// TwinCAT 3 PLC project GetConnectionInfo
// ProgramVersion: 3.1.0.5
// libraries:
//   Tc2_FTP,newest,Beckhoff Automation GmbH
//   Tc2_Standard,newest,Beckhoff Automation GmbH
//   Tc2_System,newest,Beckhoff Automation GmbH
//   Tc3_Module,newest,Beckhoff Automation GmbH
// project tree:
//   / PlcTask.TcTTO
//   POUs/ MAIN.TcPOU
// (motion and I/O tree: see PLC project fileupload)
// real-time tasks:
//   TASK PlcTask: cycle T#10ms, priority 20, ADS port 350

CONFIGURATION GetConnectionInfo
    RESOURCE PLC ON TwinCAT3
        TASK PlcTask(INTERVAL := T#10ms, PRIORITY := 20);
        PROGRAM MAIN WITH PlcTask : MAIN;
    END_RESOURCE
END_CONFIGURATION

// ---- POUs/MAIN.TcPOU
PROGRAM MAIN
VAR
	FB_FTP_Info1	: FB_FTP_Info;
	list			: ARRAY [0..5] OF ST_FTP_ConnInfo;
	startstop		: BOOL;
	busy			: BOOL;
	err				: BOOL;
	errid			: UDINT;
	entries			: UDINT;	
END_VAR

FB_FTP_Info1(
	sNetID:= ,
	pList:= ADR(list),
	cbList:= SIZEOF(list),
	bExecute:= startstop,
	tTimeout:= T#15s,
	bBusy=> busy,
	bError=> err,
	nErrID=> errid,
	nEntries=> entries);

END_PROGRAM
